// TIA Portal V17 export
// export: Created 2025-06-25T13:13:14.8515092Z, ExportSetting WithDefaults, DisplayName Totally Integrated Automation Portal, DisplayVersion V17 Update 8, DisplayName TIA Portal Openness, DisplayVersion V17 Update 8, DisplayName TIA Portal Version Control Interface, DisplayVersion V17, DisplayName STEP 7 Professional, DisplayVersion V17 Update 8, DisplayName STEP 7 Safety, DisplayVersion V17 Update 6, DisplayName WinCC Advanced, DisplayVersion V17 Update 8
FUNCTION_BLOCK "fbACS880"   // FB22, FBD
TITLE = Interface block for ABB ACS880
{ S7_Optimized_Access := 'TRUE' }
AUTHOR : Heaten
VERSION : 0.1
// stored: AutoNumber true, IsIECCheckEnabled false, IsRetainMemResEnabled false, MemoryReserve 0, SetENOAutomatically false, UDAEnableTagReadback false
   VAR_INPUT
      bCommOk : Bool;   // 0 = comm fail
      bEmergencyStop : Bool;   // 1 = E-stop, 0 = ok
      fSpeedSetpoint : Real;   // rpm
      fTorqueSetpoint : Real;   // %
      sRxInstance : "stABB_ACSx80_Rx";   // Input data raw
   END_VAR
   VAR_OUTPUT
      sTxInstance : "stABB_ACSx80_Tx";   // Output data raw
   END_VAR
   VAR_IN_OUT
      sTag : "stInverterDrive";   // This drive
   END_VAR
   VAR
      ResetTimer : TP_TIME;   // NB: Pulse timer!
   END_VAR
   VAR_TEMP
      Dummy : Real;
      Speed : Int;
      Torque : Int;
   END_VAR
BEGIN

REGION Network 1: Fieldbus comm ok
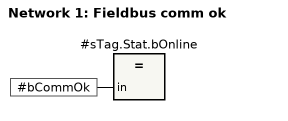
   #sTag.Stat.bOnline := #bCommOk;
END_REGION

REGION Network 2 (SCL): Data processing: READ
   // handle Act1 & Act2
   "fcAnalogInput"(bValidData := #bCommOk, iAI := WORD_TO_INT(#sRxInstance.Act1), fOffset := 0.0, sTag := #sTag.Stat.Speed, fEngValue => #Dummy);
   "fcAnalogInput"(bValidData := #bCommOk, iAI := WORD_TO_INT(#sRxInstance.Act2), fOffset := 0.0, sTag := #sTag.Stat.Torque, fEngValue => #Dummy);
   "fcAnalogInput"(bValidData := #bCommOk, iAI := WORD_TO_INT(#sRxInstance.DataIO_12), fOffset := 0.0, sTag := #sTag.Stat.Power, fEngValue => #Dummy);

   // Status Word
   IF #bCommOk = FALSE THEN
       // Zero out all data on comm error
       #sTag.Stat.bRemote := FALSE;
       #sTag.Stat.bRun := FALSE;
       #sTag.Stat.bTrip := FALSE;
       #sTag.Stat.bReady := FALSE;
   ELSE
       // Status Word (ABB Drives profile)
       // BIT  NAME            STATE
       // 0    RDY_ON          Ready to Switch On
       // 1    RDY_RUN         0 = OFF1 active, 1 = Ready to operate
       // 2    RDY_REF         Operation enabled
       // 3    TRIPPED         Fault
       // 4    OFF_2_STATUS    0 = OFF2 active, 1 = OFF2 inactive
       // 5    OFF_3_STATUS    0 = OFF3 active, 1 = OFF3 inactive
       // 6    SWC_ON_INHIB    1 = Switch-on inhibited
       // 7    ALARM           0 = No warning/alarm, 1 = warning/alarm
       // 8    AT_SETPOINT     1 = actual value within tolerance of Ref
       // 9    REMOTE          0 = local control 1 = remote control
       // 10   ABOVE_LIMIT     1 = actual speed >= supervision limit
       // 11   USER_0          
       // 12   USER_1
       // 13   USER_2
       // 14   USER_3
       // 15   Reserved by ABB
       #sTag.Stat.bReady := #sRxInstance.SW.%X0;
       #sTag.Stat.bRun := #sRxInstance.SW.%X2;
       #sTag.Stat.bTrip := #sRxInstance.SW.%X3;
       #sTag.Stat.bRemote := #sRxInstance.SW.%X9;

       // Further optional processing based on variant
       CASE #sTag.nVariant OF
           0 : ;
           1 : ;
       END_CASE;
   END_IF;
END_REGION

REGION Network 3 (SCL): Data processing: WRITE
   // Outputs get written even if there is comm error
   // Control Word (ABB Drives profile)
   // BIT  NAME            STATE
   // 0    OFF1_CONTROL    0 = OFF1 Active, 1 = Proceed to READY TO OPERATE
   // 1    OFF2_CONTROL    0 = OFF2 Active, 1 = Continue operation
   // 2    OFF3_CONTROL    0 = OFF3 Active, 1 = Continue operation
   // 3    INHIBIT_OPERATION 0 = inhibit, 1 = Proceed to OPERATION ENABLED (Run?)
   // 4    RAMP_OUT_ZERO   0 = force ramp output to zero, 1 = normal operation
   // 5    RAMP_HOLD       0 = halt ramping (hold output), 1 = normal operation
   // 6    RAMP_IN_ZERO    0 = force ramp input to zero, 1 = normal operation
   // 7    RESET           0 = normal operation, 1 = reset fault
   // 8    JOGGING_1       0 = normal operation, 1 = run at Jogging 1 speed
   // 9    JOGGING_2       0 = normal operation, 1 = run at Jogging 2 speed
   // 10   REMOTE_CMD      0 = ?, 1 = fieldbus controlled
   // 11   EXT_CTRL_LOC    0 = EXT1, 1 = EXT2
   // 12   USER_0
   // 13   USER_1
   // 14   USER_2
   // 15   USER_3
   // NOTE: the firmware manual describes a state machine for starting the drive. But the transitions from
   // one state to another are levels and not edges, therefore several conditions can be combined and sent
   // at the same time.
   // Stop : CW = 16#0476
   // Ready : CW = 16#47E
   // Run  : CW = 16#047F
   // Reset: CW = 16#04F6
   // NOTE 2: sTag.Cmd.bReady is for enabling the drive without running it; sTag.Cmd.bRun will override this, so don't use bReady to turn the drive on and off

   // Make reset a pulse
   #ResetTimer(IN := #sTag.Cmd.bReset, PT := T#3s);

   // Control word
   IF #bEmergencyStop = TRUE THEN
       #sTxInstance.CW := 16#0476;
   ELSIF #ResetTimer.Q THEN
       #sTxInstance.CW := 16#04F6;
       #sTag.Cmd.bReset := FALSE;
   ELSIF #sTag.Cmd.bManualRun = TRUE AND #sTag.Cmd.bManualMode = TRUE THEN
       #sTxInstance.CW := 16#047F;
   ELSIF #sTag.Cmd.bRun = TRUE THEN
       #sTxInstance.CW := 16#047F;
   ELSIF #sTag.Cmd.bReady = TRUE THEN
       #sTxInstance.CW := 16#047E;
   ELSE
       #sTxInstance.CW := 16#0476;
   END_IF;

   // Setpoints
   IF #bEmergencyStop = TRUE THEN
       "fcCalcAssign"(fValue := 0.0, sTag := #sTag.Cmd.Speed.Eng);
       "fcCalcAssign"(fValue := 0.0, sTag := #sTag.Cmd.Torque.Eng);
       #sTag.Cmd.bManualMode := FALSE;
       #sTag.Cmd.fManualSpeed := 0.0;
   ELSIF #sTag.Cmd.bManualMode = TRUE THEN
       "fcCalcAssign"(fValue := #sTag.Cmd.fManualSpeed, sTag:= #sTag.Cmd.Speed.Eng);
       "fcCalcAssign"(fValue := #sTag.Cmd.fManualTorque, sTag := #sTag.Cmd.Torque.Eng);
   ELSE
       // Allow Manual Mode to take over from auto in run state and with same setpoints
       IF #sTag.Stat.bRun = TRUE THEN
           #sTag.Cmd.bManualRun := #sTag.Cmd.bRun;
           #sTag.Cmd.fManualSpeed := #sTag.Cmd.Speed.Eng.fValue;
           #sTag.Cmd.fManualTorque := #sTag.Cmd.Torque.Eng.fValue;
       END_IF;

       "fcCalcAssign"(fValue := #fSpeedSetpoint, sTag:= #sTag.Cmd.Speed.Eng);
       "fcCalcAssign"(fValue := #fTorqueSetpoint, sTag := #sTag.Cmd.Torque.Eng);
   END_IF;

   // Write to fieldbus
   "fcAnalogOutput"(bOutputOk := #bCommOk, sTag := #sTag.Cmd.Speed, iAO => #Speed);
   "fcAnalogOutput"(bOutputOk := #bCommOk, sTag := #sTag.Cmd.Torque, iAO => #Torque);

   #sTxInstance.Ref1 := INT_TO_WORD(#Speed);
   #sTxInstance.Ref2 := INT_TO_WORD(#Torque);
END_REGION
END_FUNCTION_BLOCK
